	              // Calculate end point for circle mode 0 by given mode 0
	              #tempRetValue := "LKinCtrl_CalcCircTangOrthPathPlane"(circlePoint := #tempNextCmdIn.endPoint,
	                                                                    circleCenterPoint := #tempNextCmdIn.circleCenterPoint,
	                                                                    pathPlane := #pathPlane,
	                                                                    compDirection := #compensationDirection,
	                                                                    pathChoice := #tempNextCmdIn.pathChoice,
	                                                                    vUnitTangentialPathPlane => #tempNextCmdOut.tangentialUnitVecEnd,
	                                                                    vUnitOrthogonalPathPlane => #tempNextCmdOut.orthogonalUnitVecEnd);

	              IF (#tempRetValue <> 0) THEN
	                #LKinCtrl_OffsetContour.returnValue := #tempRetValue;
	                #LKinCtrl_OffsetContour."region" := #COFF_REGION_TYPE_RAD_COMP_CIRC_NONE;
	                #LKinCtrl_OffsetContour.subBlockNumber := 35056;
	                #LKinCtrl_OffsetContour.internalNumber := 450;
	                RETURN;
	              END_IF;

	              // Scale othogonal vector with tool radius to get orthogonal shift
	              #tempNextCmdOut.orthogonalShiftEnd := "LKinCtrl_VecScale"(vIn := #tempNextCmdOut.orthogonalUnitVecEnd,
	                                                                        factor := #toolRadius);


	              #tempNextCmdOut.endPoint := "LKinCtrl_VecAdd"(vIn1 := #tempNextCmdIn.endPoint,
	                                                            vIn2 := #tempNextCmdOut.orthogonalShiftEnd);
	            ELSIF (#tempNextCmdIn.circleMode = "CM_CENTER") THEN
	              (*
	              // Calculate end point for circle mode 0 by given mode 1
	              #tempRetValue := "LKinCtrl_CalcCircEndPointWithGivenCenterAndAngle"(circleStartPoint := #tempCurrentPointRadComp,
	                                                                                  circleCenterPoint := #tempNextCmdIn.circleCenterPoint,
	                                                                                  pathPlane := #pathPlane,
	                                                                                  pathChoice := #tempNextCmdIn.pathChoice,
	                                                                                  angle := #tempNextCmdIn.circleAngle,
	                                                                                  endPoint => #tempNextCmdOut.endPoint);

	              IF (#tempRetValue <> 0) THEN
	                #LKinCtrl_OffsetContour.returnValue := #tempRetValue;
	                #LKinCtrl_OffsetContour."region" := #COFF_REGION_TYPE_RAD_COMP_CIRC_NONE;
	                #LKinCtrl_OffsetContour.subBlockNumber := 35053;
	                #LKinCtrl_OffsetContour.internalNumber := 451;
	                RETURN;
	              END_IF;
	              *)
	              // Calculate end point for circle mode 0 by given mode 0
	              #tempRetValue := "LKinCtrl_CalcCircTangOrthPathPlane"(circlePoint := #tempNextCmdIn.endPoint,
	                                                                    circleCenterPoint := #tempNextCmdIn.circleCenterPoint,
	                                                                    pathPlane := #pathPlane,
	                                                                    compDirection := #compensationDirection,
	                                                                    pathChoice := #tempNextCmdIn.pathChoice,
	                                                                    vUnitTangentialPathPlane => #tempNextCmdOut.tangentialUnitVecEnd,
	                                                                    vUnitOrthogonalPathPlane => #tempNextCmdOut.orthogonalUnitVecEnd);

	              IF (#tempRetValue <> 0) THEN
	                #LKinCtrl_OffsetContour.returnValue := #tempRetValue;
	                #LKinCtrl_OffsetContour."region" := #COFF_REGION_TYPE_RAD_COMP_CIRC_NONE;
	                #LKinCtrl_OffsetContour.subBlockNumber := 35056;
	                #LKinCtrl_OffsetContour.internalNumber := 450;
	                RETURN;
	              END_IF;

	              // Scale othogonal vector with tool radius to get orthogonal shift
	              #tempNextCmdOut.orthogonalShiftEnd := "LKinCtrl_VecScale"(vIn := #tempNextCmdOut.orthogonalUnitVecEnd,
	                                                                        factor := #toolRadius);


	              #tempNextCmdOut.endPoint := "LKinCtrl_VecAdd"(vIn1 := #tempNextCmdIn.endPoint,
	                                                            vIn2 := #tempNextCmdOut.orthogonalShiftEnd);

	            ELSIF (#tempNextCmdIn.circleMode = "CM_RADIUS") THEN
	              (*
	              // ------------ Via the circle radius and the end point in a main plane ("CircMode" = 2) ------------
	              // Calculate angle between center/start and center/end of circle - always the smaller one!!!
	              #tempRetValue := "LKinCtrl_CalcAngleBetweenVectors"(point1 := #tempCurrentPointRadComp,//#tempNextCmdOut.startPointOrthShifted,
	                                                                  point2 := #tempNextCmdIn.endPoint,//#tempNextCmdOut.endPoint,
	                                                                  intersectionPoint := #tempNextCmdIn.circleCenterPoint,
	                                                                  angle => #tempAngle);

	              IF (#tempRetValue <> 0) THEN
	                #LKinCtrl_OffsetContour.returnValue := #tempRetValue;
	                #LKinCtrl_OffsetContour."region" := #COFF_REGION_TYPE_RAD_COMP_CIRC_NONE;
	                #LKinCtrl_OffsetContour.subBlockNumber := 35059;
	                #LKinCtrl_OffsetContour.internalNumber := 452;
	                RETURN;
	              END_IF;

	              // Calculate end point for circle mode 0 by given mode 2
	              #tempRetValue := "LKinCtrl_CalcCircEndPointWithGivenCenterAndAngle"(circleStartPoint := #tempCurrentPointRadComp, //tempNextCmdOut.startPointOrthShifted,
	                                                                                  circleCenterPoint := #tempNextCmdIn.circleCenterPoint,
	                                                                                  pathPlane := #pathPlane,
	                                                                                  pathChoice := #tempNextCmdIn.pathChoice,
	                                                                                  angle := #tempAngle,
	                                                                                  endPoint => #tempNextCmdOut.endPoint);



	              IF (#tempRetValue <> 0) THEN
	                #LKinCtrl_OffsetContour.returnValue := #tempRetValue;
	                #LKinCtrl_OffsetContour."region" := #COFF_REGION_TYPE_RAD_COMP_CIRC_NONE;
	                #LKinCtrl_OffsetContour.subBlockNumber := 35053;
	                #LKinCtrl_OffsetContour.internalNumber := 453;
	                RETURN;
	              END_IF;
	              *)
	              ;
	            END_IF;
	            *)

	          END_REGION
	        END_IF;


	        // ############# M O D I F Y   N E X T   C I R C U L A R   C O M M A N D   #############
	        REGION Modify next circular command
	          // Distinguish between different circular modes
	          IF (#tempNextCmdIn.circleMode = "CM_BORDER") THEN

	            // ------------ Via an intermediate point and the end point ("CircMode" = 0) ------------
	            // Calculate intermediate point for circle mode 0 by given mode 0
	            // Calculate circle paramters
	            #tempRetValue := "LKinCtrl_CalcCircTangOrthPathPlane"(circlePoint := #tempNextCmdIn.circleIntermediatePoint,
	                                                                  circleCenterPoint := #tempNextCmdIn.circleCenterPoint,
	                                                                  pathPlane := #pathPlane,
	                                                                  compDirection := #compensationDirection,
	                                                                  pathChoice := #tempNextCmdIn.pathChoice,
	                                                                  vUnitTangentialPathPlane => #tempNextCmdOut.tangentialUnitVecIntermediate,
	                                                                  vUnitOrthogonalPathPlane => #tempNextCmdOut.orthogonalUnitVecIntermediate);

	            IF (#tempRetValue <> 0) THEN
	              #LKinCtrl_OffsetContour.returnValue := #tempRetValue;
	              #LKinCtrl_OffsetContour."region" := #COFF_REGION_TYPE_RAD_COMP_CIRC_GEN;
	              #LKinCtrl_OffsetContour.subBlockNumber := 35056;
	              #LKinCtrl_OffsetContour.internalNumber := 460;
	              RETURN;
	            END_IF;

	            // Scale othogonal vector with tool radius to get orthogonal shift
	            #tempNextCmdOut.orthogonalShiftIntermediate := "LKinCtrl_VecScale"(vIn := #tempNextCmdOut.orthogonalUnitVecIntermediate,
	                                                                               factor := #toolRadius);


	            #tempNextCmdOut.circleIntermediatePoint := "LKinCtrl_VecAdd"(vIn1 := #tempNextCmdIn.circleIntermediatePoint,
	                                                                         vIn2 := #tempNextCmdOut.orthogonalShiftIntermediate);

	            // Change circle mode to 0 - intermediate point and the end point ("CircMode" = 0)
	            #tempNextCmdOut.circleMode := "CM_BORDER";

	          ELSIF (#tempNextCmdIn.circleMode = "CM_CENTER") THEN

	            // Take care of greater angles
	            // #tempMod := TRUNC(#tempNextCmdIn.circleAngle / 180.0);
	            // IF (#tempMod >= 3) THEN
	            //   #tempAngle := #tempNextCmdIn.circleAngle - ((#tempMod - 1) * 180);
	            // ELSE
	            //   #tempAngle := #tempNextCmdIn.circleAngle;
	            // END_IF;

	            // V01.02.02
	            // Calculate compensated angle
	            #tempRetValue := "LKinCtrl_CalcAngleBetweenVectors"(point1 := #tempCurrentPointRadComp, //tempNextCmdOut.startPointOrthShifted,
	                                                                point2 := #tempNextCmdOut.endPoint,
	                                                                intersectionPoint := #tempNextCmdIn.circleCenterPoint,
	                                                                angle => #tempAngle);

	            IF (#tempRetValue <> 0) THEN
	              #LKinCtrl_OffsetContour.returnValue := #tempRetValue;
	              #LKinCtrl_OffsetContour."region" := #COFF_REGION_TYPE_RAD_COMP_CIRC_GEN;
	              #LKinCtrl_OffsetContour.subBlockNumber := 35059;
	              #LKinCtrl_OffsetContour.internalNumber := 461;
	              RETURN;
	            END_IF;
	            //
	            // Calculate intermediate point for circle mode 0 by given mode 1
	            #tempRetValue := "LKinCtrl_CalcCircEndPointWithGivenCenterAndAngle"(circleStartPoint := #tempCurrentPointRadComp, // tempNextCmdOut.startPointOrthShifted,
	                                                                                circleCenterPoint := #tempNextCmdIn.circleCenterPoint,
	                                                                                pathPlane := #pathPlane,
	                                                                                pathChoice := #tempNextCmdIn.pathChoice,
	                                                                                angle := #tempAngle / 2.0,//(#tempNextCmdIn.circleAngle / 2.0),
	                                                                                endPoint => #tempNextCmdOut.circleIntermediatePoint);
	            IF (#tempRetValue <> 0) THEN
	              #LKinCtrl_OffsetContour.returnValue := #tempRetValue;
	              #LKinCtrl_OffsetContour."region" := #COFF_REGION_TYPE_RAD_COMP_CIRC_GEN;
	              #LKinCtrl_OffsetContour.subBlockNumber := 35053;
	              #LKinCtrl_OffsetContour.internalNumber := 462;
	              RETURN;
	            END_IF;

	            // Ceck if resulting path choice (circle with intermediate point) has changed --> circle larger than 360°
	            // Calculate path choice
	            #tempRetValue := "LKinCtrl_CalcCircPathChoiceByIntermediatePointAndEndPoint"(circleStartPoint := #tempCurrentPointRadComp, //tempNextCmdOut.startPointOrthShifted,
	                                                                                         circleEndPoint := #tempNextCmdOut.endPoint,
	                                                                                         circleintermediatePoint := #tempNextCmdOut.circleIntermediatePoint,
	                                                                                         pathPlane := #pathPlane,
	                                                                                         pathChoice => #tempPathChoice);


	            IF (#tempRetValue <> 0) THEN
	              #LKinCtrl_OffsetContour.returnValue := #tempRetValue;
	              #LKinCtrl_OffsetContour."region" := #COFF_REGION_TYPE_RAD_COMP_CIRC_GEN;
	              #LKinCtrl_OffsetContour.subBlockNumber := 35058;
	              #LKinCtrl_OffsetContour.internalNumber := 463;
	              RETURN;
	            END_IF;

	            IF ((#tempNextCmdIn.pathChoice <> #tempPathChoice) OR
	              (#tempNextCmdIn.circleAngle >= 360.0))
	            THEN

	              // V01.02.02 - done before now
	              // // Calculate additional angle between center/start and center/end of circle - always the smaller one!!!
	              // #tempRetValue := "LKinCtrl_CalcAngleBetweenVectors"(point1 := #tempCurrentPointRadComp, //tempNextCmdOut.startPointOrthShifted,
	              //                                                     point2 := #tempNextCmdOut.endPoint,
	              //                                                     intersectionPoint := #tempNextCmdIn.circleCenterPoint,
	              //                                                     angle => #tempAngle);

	              // IF (#tempRetValue <> 0) THEN
	              //   #LKinCtrl_OffsetContour.returnValue := #tempRetValue;
	              //   #LKinCtrl_OffsetContour."region" := #COFF_REGION_TYPE_RAD_COMP_CIRC_GEN;
	              //   #LKinCtrl_OffsetContour.subBlockNumber := 35059;
	              //   #LKinCtrl_OffsetContour.internalNumber := 463;
	              //   RETURN;
	              // END_IF;

	              // Circle > 360° - not possible with circle type border
	              IF (#tempNextCmdIn.pathChoice <> #tempPathChoice) THEN
	                #tempNextCmdOut.circleAngle := (TRUNC((#tempNextCmdIn.circleAngle + 180.0) / 360.0) * 360.0) + #tempAngle;
	              ELSE
	                #tempNextCmdOut.circleAngle := (TRUNC((#tempNextCmdIn.circleAngle + 180.0) / 360.0) * 360.0) - #tempAngle;
	              END_IF;

	              #tempNextCmdOut.circleMode := "CM_CENTER";
	            ELSE

	              // V01.02.02
	              // Output angle - for debugging only
	              #tempNextCmdOut.circleAngle := #tempAngle;

	              // Change circle mode to 0 - intermediate point and the end point ("CircMode" = 0)
	              #tempNextCmdOut.circleMode := "CM_BORDER";
	            END_IF;

	          ELSIF (#tempNextCmdIn.circleMode = "CM_RADIUS") THEN
	            // ------------ Via the circle radius and the end point in a main plane ("CircMode" = 2) ------------
	            // Calculate angle between center/start and center/end of circle - always the smaller one!!!
	            #tempRetValue := "LKinCtrl_CalcAngleBetweenVectors"(point1 := #tempCurrentPointRadComp,
	                                                                point2 := #tempNextCmdOut.endPoint,
	                                                                intersectionPoint := #tempNextCmdIn.circleCenterPoint,
	                                                                angle => #tempAngle);

	            IF (#tempRetValue <> 0) THEN
	              #LKinCtrl_OffsetContour.returnValue := #tempRetValue;
	              #LKinCtrl_OffsetContour."region" := #COFF_REGION_TYPE_RAD_COMP_CIRC_GEN;
	              #LKinCtrl_OffsetContour.subBlockNumber := 35059;
	              #LKinCtrl_OffsetContour.internalNumber := 464;
	              RETURN;
	            END_IF;

	            // Calculate intermediate point for circle mode 0 by given mode 2
	            #tempRetValue := "LKinCtrl_CalcCircEndPointWithGivenCenterAndAngle"(circleStartPoint := #tempCurrentPointRadComp, //tempNextCmdOut.startPointOrthShifted,
	                                                                                circleCenterPoint := #tempNextCmdIn.circleCenterPoint,
	                                                                                pathPlane := #pathPlane,
	                                                                                pathChoice := #tempNextCmdIn.pathChoice,
	                                                                                angle := (#tempAngle / 2.0),
	                                                                                endPoint => #tempNextCmdOut.circleIntermediatePoint);

	            IF (#tempRetValue <> 0) THEN
	              #LKinCtrl_OffsetContour.returnValue := #tempRetValue;
	              #LKinCtrl_OffsetContour."region" := #COFF_REGION_TYPE_RAD_COMP_CIRC_GEN;
	              #LKinCtrl_OffsetContour.subBlockNumber := 35053;
	              #LKinCtrl_OffsetContour.internalNumber := 465;
	              RETURN;
	            END_IF;

	            // Change circle mode to 0 - intermediate point and the end point ("CircMode" = 0)
	            #tempNextCmdOut.circleMode := "CM_BORDER";

	          END_IF;

	          // Additional check - has the direction between start - end and start - compensated end changed
	          // --> Reversal path with "small" length (and "large" tool radius) leads to unexpected circle (mathematical correct but in an unexpected direction)
	          REGION Additional plausibility check
	            #tempRetValue := "LKinCtrl_CalcAngleBetweenVectors"(point1 := #tempNextCmdOut.endPoint,
	                                                                point2 := #tempNextCmdIn.endPoint,
	                                                                intersectionPoint := #tempCurrentPoint,
	                                                                angle => #tempAngle);

	            IF (#tempRetValue <> 0) THEN
	              #LKinCtrl_OffsetContour.returnValue := #tempRetValue;
	              #LKinCtrl_OffsetContour."region" := #COFF_REGION_TYPE_RAD_COMP_CIRC_GEN;
	              #LKinCtrl_OffsetContour.subBlockNumber := 35059;
	              #LKinCtrl_OffsetContour.internalNumber := 470;
	              RETURN;
	            END_IF;

	            IF ((#tempAngle > #COFF_CIRC_REVERSAL_TOLERANCE_ANGLE) AND
	              ("LKinCtrl_VecAbs"("LKinCtrl_VecSub"(vIn1 := #tempNextCmdOut.endPoint,
	                                                                      vIn2 := #tempNextCmdOut.circleIntermediatePoint)) < (2.0 * #toolRadius)))
	            THEN
	              #LKinCtrl_OffsetContour.returnValue := #ERR_COFF_NO_SOLUTION_FOR_GIVEN_CIRCULAR_CMD;
	              #LKinCtrl_OffsetContour."region" := #COFF_REGION_TYPE_RAD_COMP_CIRC_GEN;
	              #LKinCtrl_OffsetContour.subBlockNumber := 0;
	              #LKinCtrl_OffsetContour.internalNumber := 471;
	              RETURN;
	            END_IF;

	          END_REGION

	          // V01.02.02
	          REGION Additional plausibility check
	            // Check if circle radius has become smaller than possible - compensation inside

	            // Calculate the length end point circle center
	            #tempRetValue := "LKinCtrl_CalcVecDistancePathPlane"(vectorInA := #tempNextCmdIn.endPoint,
	                                                                 vectorInB := #tempNextCmdIn.circleCenterPoint,
	                                                                 pathPlane := #pathPlane,
	                                                                 distancePathPlane => #tempCircleDistance1);

	            IF (#tempRetValue <> 0) THEN
	              #LKinCtrl_OffsetContour.returnValue := #tempRetValue;
	              #LKinCtrl_OffsetContour."region" := #COFF_REGION_TYPE_RAD_COMP_CIRC_GEN;
	              #LKinCtrl_OffsetContour.subBlockNumber := 35067;
	              #LKinCtrl_OffsetContour.internalNumber := 472;
	              RETURN;
	            END_IF;

	            #tempRetValue := "LKinCtrl_CalcVecDistancePathPlane"(vectorInA := #tempNextCmdOut.endPoint,
	                                                                 vectorInB := #tempNextCmdIn.circleCenterPoint,
	                                                                 pathPlane := #pathPlane,
	                                                                 distancePathPlane => #tempCircleDistance2);

	            IF (#tempRetValue <> 0) THEN
	              #LKinCtrl_OffsetContour.returnValue := #tempRetValue;
	              #LKinCtrl_OffsetContour."region" := #COFF_REGION_TYPE_RAD_COMP_CIRC_GEN;
	              #LKinCtrl_OffsetContour.subBlockNumber := 35067;
	              #LKinCtrl_OffsetContour.internalNumber := 473;
	              RETURN;
	            END_IF;

	            IF (#tempCircleDistance2 < #tempCircleDistance1) THEN
	              // inside circle - check plausibility
	              // Tool radius must not be greater than circle radius
	              IF (#toolRadius > (#tempCircleDistance1 - #RADIUS_PLAUSIBLITY_TOLERANCE)) THEN
	                #LKinCtrl_OffsetContour.returnValue := #ERR_COFF_NO_SOLUTION_FOR_GIVEN_CIRCULAR_CMD;
	                #LKinCtrl_OffsetContour."region" := #COFF_REGION_TYPE_RAD_COMP_CIRC_GEN;
	                #LKinCtrl_OffsetContour.subBlockNumber := 0;
	                #LKinCtrl_OffsetContour.internalNumber := 474;
	                RETURN;
	              END_IF;
	              // Tool radius must not be greater than circle start and end point (uncompensated)
	              #tempRetValue := "LKinCtrl_CalcVecDistancePathPlane"(vectorInA := #tempCurrentPoint,
	                                                                   vectorInB := #tempNextCmdIn.endPoint,
	                                                                   pathPlane := #pathPlane,
	                                                                   distancePathPlane => #tempCircleDistance3);

	              IF (#tempRetValue <> 0) THEN
	                #LKinCtrl_OffsetContour.returnValue := #tempRetValue;
	                #LKinCtrl_OffsetContour."region" := #COFF_REGION_TYPE_RAD_COMP_CIRC_GEN;
	                #LKinCtrl_OffsetContour.subBlockNumber := 35067;
	                #LKinCtrl_OffsetContour.internalNumber := 475;
	                RETURN;
	              END_IF;

	              IF (#toolRadius > (#tempCircleDistance3 - #RADIUS_PLAUSIBLITY_TOLERANCE)) THEN
	                #LKinCtrl_OffsetContour.returnValue := #ERR_COFF_NO_SOLUTION_FOR_GIVEN_CIRCULAR_CMD;
	                #LKinCtrl_OffsetContour."region" := #COFF_REGION_TYPE_RAD_COMP_CIRC_GEN;
	                #LKinCtrl_OffsetContour.subBlockNumber := 0;
	                #LKinCtrl_OffsetContour.internalNumber := 476;
	                RETURN;
	              END_IF;

	            END_IF;

	          END_REGION
	        END_REGION
	      END_IF;
	    END_REGION

	  END_IF;

	  // V01.00.01
	  // Output before length compensation
	  #nextPositionAbsoluteRadCompOut := "LKinCtrl_3DPointToCartesianCoord"(#tempNextCmdOut.endPoint);
	END_REGION TOOL_RADIUS_COMPENSATION

	// Tool length compensation
	REGION TOOL_LENGTH_COMPENSATION
	  IF (#tempToolLengthComp) THEN
	    // Next command
	    // -------------------------------------------------------------------------------------
	    // Compensate coordinates of according to path plane
	    // End point
	    #tempRetValue := "LKinCtrl_CalcToolLengthCompensation"(toolLength := #toolLength,
	                                                           pathPlane := #pathPlane,
	                                                           point := #tempNextCmdOut.endPoint);
	    IF (#tempRetValue <> 0) THEN
	      #LKinCtrl_OffsetContour.returnValue := #tempRetValue;
	      #LKinCtrl_OffsetContour."region" := #COFF_REGION_TYPE_LEN_COMP_NEXT;
	      #LKinCtrl_OffsetContour.subBlockNumber := 35070;
	      #LKinCtrl_OffsetContour.internalNumber := 601;
	      RETURN;
	    END_IF;

	    // Circle coordinates
	    IF (#tempNextCmdOut.cmdType = "LKINCTRL_MC_MOVECIRCULARABS") THEN

	      IF (#tempNextCmdOut.circleMode = "CM_BORDER") THEN

	        #tempRetValue := "LKinCtrl_CalcToolLengthCompensation"(toolLength := #toolLength,
	                                                               pathPlane := #pathPlane,
	                                                               point := #tempNextCmdOut.circleIntermediatePoint);
	        IF (#tempRetValue <> 0) THEN
	          #LKinCtrl_OffsetContour.returnValue := #tempRetValue;
	          #LKinCtrl_OffsetContour."region" := #COFF_REGION_TYPE_LEN_COMP_NEXT;
	          #LKinCtrl_OffsetContour.subBlockNumber := 35070;
	          #LKinCtrl_OffsetContour.internalNumber := 602;
	          RETURN;
	        END_IF;

	      ELSIF (#tempNextCmdOut.circleMode = "CM_CENTER") THEN

	        #tempRetValue := "LKinCtrl_CalcToolLengthCompensation"(toolLength := #toolLength,
	                                                               pathPlane := #pathPlane,
	                                                               point := #tempNextCmdOut.circleCenterPoint);
	        IF (#tempRetValue <> 0) THEN
	          #LKinCtrl_OffsetContour.returnValue := #tempRetValue;
	          #LKinCtrl_OffsetContour."region" := #COFF_REGION_TYPE_LEN_COMP_NEXT;
	          #LKinCtrl_OffsetContour.subBlockNumber := 35070;
	          #LKinCtrl_OffsetContour.internalNumber := 603;
	          RETURN;
	        END_IF;

	      ELSIF (#tempNextCmdOut.circleMode = "CM_RADIUS") THEN
	        ;
	      ELSE
	        #LKinCtrl_OffsetContour.returnValue := #ERR_COFF_INTERNAL; // Internal error
	        #LKinCtrl_OffsetContour."region" := #COFF_REGION_TYPE_LEN_COMP_NEXT;
	        #LKinCtrl_OffsetContour.internalNumber := 604;
	        RETURN;
	      END_IF;
	    END_IF;

	    // Intermediate command
	    // -------------------------------------------------------------------------------------
	    // Compensate coordinates of according to path plane
	    IF (#tempIntermediateCmdOut.cmdType <> -1) THEN

	      // End point
	      #tempRetValue := "LKinCtrl_CalcToolLengthCompensation"(toolLength := #toolLength,
	                                                             pathPlane := #pathPlane,
	                                                             point := #tempIntermediateCmdOut.endPoint);
	      IF (#tempRetValue <> 0) THEN
	        #LKinCtrl_OffsetContour.returnValue := #tempRetValue;
	        #LKinCtrl_OffsetContour."region" := #COFF_REGION_TYPE_LEN_COMP_INTER_CMD;
	        #LKinCtrl_OffsetContour.subBlockNumber := 35070;
	        #LKinCtrl_OffsetContour.internalNumber := 605;
	        RETURN;
	      END_IF;

	      // Always circle by intemdiate point and end point
	      #tempRetValue := "LKinCtrl_CalcToolLengthCompensation"(toolLength := #toolLength,
	                                                             pathPlane := #pathPlane,
	                                                             point := #tempIntermediateCmdOut.circleIntermediatePoint);
	      IF (#tempRetValue <> 0) THEN
	        #LKinCtrl_OffsetContour.returnValue := #tempRetValue;
	        #LKinCtrl_OffsetContour."region" := #COFF_REGION_TYPE_LEN_COMP_INTER_CMD;
	        #LKinCtrl_OffsetContour.subBlockNumber := 35070;
	        #LKinCtrl_OffsetContour.internalNumber := 606;
	        RETURN;
	      END_IF;
	    END_IF;

	    // Next but one command - not needed - no output
	    // -------------------------------------------------------------------------------------
	    (*
	    // Compensate coordinates of according to path plane
	    // End point
	    #tempRetValue := "LKinCtrl_CalcToolLengthCompensation"(toolLength := #toolLength,
	                                                           pathPlane := #pathPlane,
	                                                           point := #tempNextButOneCmdOut.endPoint);
	    IF (#tempRetValue <> 0) THEN
	      #LKinCtrl_OffsetContour.returnValue := #tempRetValue;
	      #LKinCtrl_OffsetContour."region" := #COFF_REGION_TYPE_LEN_COMP_NEXT_BUT_ONE_CMD;
	      #LKinCtrl_OffsetContour.subBlockNumber := 35070;
	      #LKinCtrl_OffsetContour.internalNumber := 607
	      RETURN;
	    END_IF;
	    *)
	  END_IF;
	END_REGION

	REGION Output data

	  // ############# O U T P U T   D A T A  #############
	  // ######################################
	  IF (#tempToolRadiusComp OR #tempToolLengthComp) THEN
	    // Next command

	    #nextCommandOut.cmdType := #tempNextCmdOut.cmdType;
	    #nextCommandOut.cmdCoordinates.cartesianPosition := "LKinCtrl_3DPointToCartesianCoord"(#tempNextCmdOut.endPoint);

	    IF (#tempNextCmdOut.cmdType = "LKINCTRL_MC_MOVECIRCULARABS") THEN
	      #nextCommandOut.cmdParameters.circleParameters.circMode := #tempNextCmdOut.circleMode;

	      IF (#tempNextCmdOut.circleMode = "CM_BORDER") THEN
	        #nextCommandOut.cmdParameters.circleParameters.auxPoint[1] := #tempNextCmdOut.circleIntermediatePoint.x;
	        #nextCommandOut.cmdParameters.circleParameters.auxPoint[2] := #tempNextCmdOut.circleIntermediatePoint.y;
	        #nextCommandOut.cmdParameters.circleParameters.auxPoint[3] := #tempNextCmdOut.circleIntermediatePoint.z;
	        // *** AW 2022-05-29 - debugging only - compensated angle
	        #nextCommandOut.cmdParameters.circleParameters.arc := #tempNextCmdOut.circleAngle;

	      ELSIF (#tempNextCmdOut.circleMode = "CM_CENTER") THEN
	        #nextCommandOut.cmdParameters.circleParameters.pathChoice := #tempNextCmdIn.pathChoice;
	        #nextCommandOut.cmdParameters.circleParameters.circlePlane := #tempNextCmdIn.circlePlane;
	        #nextCommandOut.cmdParameters.circleParameters.auxPoint[1] := #tempNextCmdOut.circleCenterPoint.x;
	        #nextCommandOut.cmdParameters.circleParameters.auxPoint[2] := #tempNextCmdOut.circleCenterPoint.y;
	        #nextCommandOut.cmdParameters.circleParameters.auxPoint[3] := #tempNextCmdOut.circleCenterPoint.z;
	        #nextCommandOut.cmdParameters.circleParameters.arc := #tempNextCmdOut.circleAngle; // #tempNextCmdIn.circleAngle;

	      ELSIF (#tempNextCmdOut.circleMode = "CM_RADIUS") THEN
	        #nextCommandOut.cmdParameters.circleParameters.pathChoice := #tempNextCmdIn.pathChoice;
	        #nextCommandOut.cmdParameters.circleParameters.circlePlane := #tempNextCmdIn.circlePlane;
	        #nextCommandOut.cmdParameters.circleParameters.radius := #tempNextCmdIn.circleRadius;

	      ELSE
	        #LKinCtrl_OffsetContour.returnValue := #ERR_COFF_INTERNAL; // Internal error
	        #LKinCtrl_OffsetContour."region" := #COFF_REGION_TYPE_OUTPUT_DATA;
	        RETURN;
	      END_IF;
	    END_IF;

	    // Coordinate a
	    // ------------
	    // Linear absolute
	    IF (#tempNextCmdIn.cmdType = "LKINCTRL_MC_MOVELINEARABS") THEN
	      // Absolute coordinates
	      #nextCommandOut.cmdCoordinates.cartesianPosition.a := #nextCommandIn.cmdCoordinates.cartesianPosition.a;
	      // Linear relative
	    ELSIF (#tempNextCmdIn.cmdType = "LKINCTRL_MC_MOVELINEARREL") THEN
	      // Relative coordinates -> calculate absolute coordinate (always)
	      #nextCommandOut.cmdCoordinates.cartesianPosition.a := #currentPosIn.positionAbsolute.a + #nextCommandIn.cmdCoordinates.cartesianPosition.a;
	      // Circular absolute
	    ELSIF (#tempNextCmdIn.cmdType = "LKINCTRL_MC_MOVECIRCULARABS") THEN
	      // Absolute coordinates
	      #nextCommandOut.cmdCoordinates.cartesianPosition.a := #nextCommandIn.cmdCoordinates.cartesianPosition.a;
	      // Circular relative
	    ELSIF (#tempNextCmdIn.cmdType = "LKINCTRL_MC_MOVECIRCULARREL") THEN
	      // Relative coordinates -> calculate absolute coordinate (always)
	      #nextCommandOut.cmdCoordinates.cartesianPosition.a := #currentPosIn.positionAbsolute.a + #nextCommandIn.cmdCoordinates.cartesianPosition.a;
	    END_IF;

	    // Output absolute end point for next cycle (including coordinate a)
	    #nextPositionAbsoluteOut := "LKinCtrl_3DPointToCartesianCoord"(#tempNextCmdIn.endPoint);
	    #nextPositionAbsoluteOut.a := #nextCommandOut.cmdCoordinates.cartesianPosition.a;

	    // Output absolute end point (radius compensated) for next cycle (including coordinate a)
	    // V01.00.01
	    // nextPositionAbsoluteRadCompOut := "LKinCtrl_3DPointToCartesianCoord"(#tempNextCmdOut.endPoint);
	    #nextPositionAbsoluteRadCompOut.a := #nextCommandOut.cmdCoordinates.cartesianPosition.a;

	    // Intermediate command
	    IF (#tempIntermediateCmdOut.cmdType <> -1) THEN

	      // Take all parameter preliminary
	      #intermediateCommandOut := #nextCommandIn;

	      #intermediateCommandOut.cmdType := #tempIntermediateCmdOut.cmdType;
	      #intermediateCommandOut.cmdParameters.circleParameters.circMode := #tempIntermediateCmdOut.circleMode;

	      // Circle by intemdiate point and end point
	      #intermediateCommandOut.cmdCoordinates.cartesianPosition := "LKinCtrl_3DPointToCartesianCoord"(#tempIntermediateCmdOut.endPoint);
	      #intermediateCommandOut.cmdParameters.circleParameters.auxPoint[1] := #tempIntermediateCmdOut.circleIntermediatePoint.x;
	      #intermediateCommandOut.cmdParameters.circleParameters.auxPoint[2] := #tempIntermediateCmdOut.circleIntermediatePoint.y;
	      #intermediateCommandOut.cmdParameters.circleParameters.auxPoint[3] := #tempIntermediateCmdOut.circleIntermediatePoint.z;

	      // Coordinate a
	      #intermediateCommandOut.cmdCoordinates.cartesianPosition.a := #nextCommandOut.cmdCoordinates.cartesianPosition.a;
	    ELSE
	      #intermediateCommandOut.cmdType := -1;
	    END_IF;

	    // Next but one command
	    //nextButOneCommandOut.cmdType := #tempNextButOneCmdIn.cmdType;
	    //nextButOneCommandOut.cmdCoordinates.cartesianPosition := "LKinCtrl_3DPointToCartesianCoord"(#tempNextButOneCmdOut.endPoint);
	    #nextButOneCommandOut.transitionParameter[1] := #tempNextButOneCmdOut.transitionParameter1;
	  ELSE
	    // Next command
	    #nextCommandOut := #nextCommandIn;
	  END_IF;

	END_REGION

	#LKinCtrl_OffsetContour.returnValue := 16#0;
	#LKinCtrl_OffsetContour."region" := #COFF_REGION_TYPE_NONE;
	#LKinCtrl_OffsetContour.subBlockNumber := 16#0;
	#LKinCtrl_OffsetContour.internalNumber := 0;


END_FUNCTION

